PROGRAM PRG_FB_CTRL_P
VAR
	fIn								: LREAL					:= 15.0;
	fOut							: LREAL;

	eMode							: E_CTRL_MODE;
	stCTRL_P_PARAMS					: ST_CTRL_P_PARAMS;

	eErrorId						: E_CTRL_ERRORCODES;
	bError							: BOOL;

	(* controller *)
	fbCTRL_P						: FB_CTRL_P;

	bInit							: BOOL	:= TRUE;
	fbTON							: TON;
END_VAR

IF bInit THEN
	(* init parameter struct *)
	stCTRL_P_PARAMS.tCtrlCycleTime	:= T#10MS;
	stCTRL_P_PARAMS.tTaskCycleTime	:= T#10ms;
	stCTRL_P_PARAMS.fKp				:= 3;								(* gain Kp	*)

	(* set the mode to ACTIVE --> normal operation *)
	eMode	:= eCTRL_MODE_ACTIVE;

	(* reset the init flag *)
	bInit	:= FALSE;
END_IF


(* call controller *)
fbCTRL_P(fIn		:= GVL.ErrorTerm,
		 eMode		:= eMode,
		 stParams	:= stCTRL_P_PARAMS,
		 fOut		=> GVL.P_Regler,
		 eErrorId	=> eErrorId,
		 bError		=> bError);

END_PROGRAM

(* stored: Version 1.1.0.1, ProductVersion 3.1.4024.9
   POU PRG_FB_CTRL_P: Id {8237676e-ab80-4ee7-bc1d-b8d830a9c631}, SpecialFunc None *)
